FUNCTION_BLOCK FB_AxisConfig_Old
VAR_INPUT
	stConfigSet: DUT_AxisParams;
	bExecReadNC: BOOL := TRUE;
	bExecReadCoE: BOOL := TRUE;
	bExecWriteNC: BOOL := FALSE;
	bExecWriteCoe: BOOL := FALSE;
	fWriteValue: LREAL;
	nWriteIndex: INT;
END_VAR
VAR_OUTPUT
	stConfig: DUT_AxisParams;
	nErrId: UDINT;
	bErr: BOOL;
	bHasInit: BOOL;
END_VAR
VAR_IN_OUT
	Axis: AXIS_REF;
END_VAR
VAR
	fbNCRead: MC_ReadParameterSet;
	fbNCWrite: MC_WriteParameter;
	fbExecuteRiseEdge: R_Trig;
	stNC: ST_AxisParameterSet;
	stDriveRef: ST_DriveRef;
	fbReadCurrLim: FB_CoERead_ByDriveRef;
	nCurrLim: UINT;
	bCurrErr: BOOL;
	nAdsErr: UINT;
	nCANErr: UINT;
	nCount: UINT := 0;
	bErrReset: BOOL;
	fbWriteCurrLim: FB_CoeWrite_ByDriveRef;
END_VAR

// Read NC params on first cycle and after each write
// Stuff into NC object
fbNCRead(Execute:=bExecReadNC,
	Parameter:=stNC,
	Axis:=Axis);
IF bExecReadNC AND fbNCRead.Done THEN
	bExecReadNC := FALSE;
END_IF
// Translate key params to stDriveRef (different attribute names)
stDriveRef.sNetId := stNC.sAmsNetId;
stDriveRef.nSlaveAddr := stNC.nPort;
stDriveRef.nDriveNo := WORD_TO_BYTE(stNC.nChnNo);

// Read CoE params
fbReadCurrLim(bExecute:=bExecReadCoE,
	stDriveRef:=stDriveRef,
	nIndex:=16#8010,
	nSubIndex:=1,
	pDstBuf:=ADR(nCurrLim),
	cbBufLen:=SIZEOF(nCurrLim),
	bError=>bCurrErr,
	iAdsErrId=>nAdsErr,
	iCANopenErrId=>nCANErr);
IF bExecReadCoE AND NOT fbReadCurrLim.bBusy THEN
	bExecReadCoE := FALSE;
END_IF

// Write if someone flipped the write bit
fbNCWrite(Execute:=bExecWriteNC,
	ParameterNumber:=nWriteIndex,
	Value:=fWriteValue,
	Axis:=Axis,
	Error=>bErr,
	ErrorID=>nErrId);
IF bErrReset THEN
	bExecWriteNC := FALSE;
	bErrReset := FALSE;
END_IF
// Flip the write bit back and schedule a read once done writing
fbExecuteRiseEdge(CLK:=fbNCWrite.Done);
IF fbExecuteRiseEdge.Q THEN
	bExecReadNC := TRUE;
	bExecWriteNC := FALSE;
END_IF

// Write max current param
fbWriteCurrLim(bExecute:=bExecWriteCoE,
	stDriveRef:=stDriveRef,
	nIndex:=16#8010,
	nSubIndex:=1,
	pSrcBuf:=ADR(nCurrLim),
	cbBufLen:=SIZEOF(nCurrLim),
	bError=>bCurrErr,
	iAdsErrId=>nAdsErr,
	iCANopenErrId=>nCANErr);
IF bExecWriteCoE AND NOT fbWriteCurrLim.bBusy THEN
	bExecWriteCoE := FALSE;
	bExecReadCoE := TRUE;
END_IF
*)

END_FUNCTION_BLOCK

(* stored: Version 1.1.0.1, ProductVersion 3.1.4022.12
   POU FB_AxisConfig_Old: Id {13c2a29c-c79d-423f-9560-f54711b0e7b3}, SpecialFunc None *)
